ABB RAPID module: FSNH0464.mod

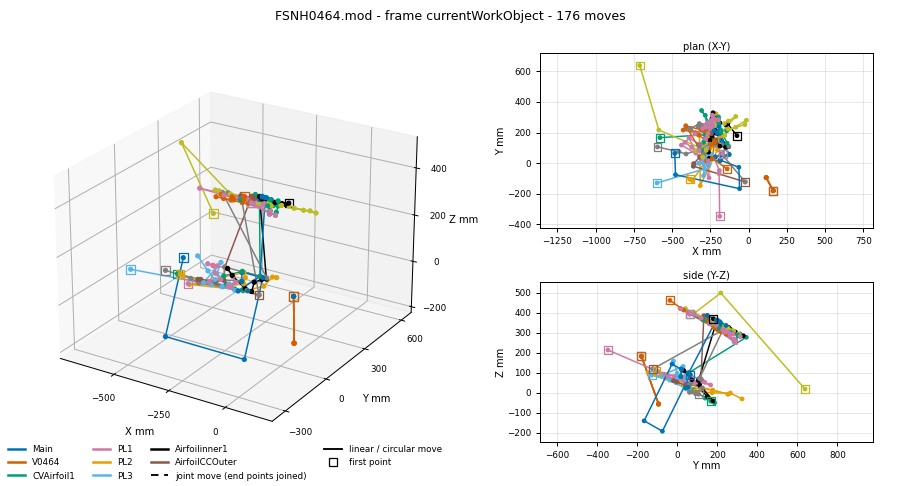
[picture p0: tool path of FSNH0464.mod in frame currentWorkObject, 176 of 176 moves have a stored position in this frame; points joined in program order, loops and branches not executed]
MODULE FSNH0464
    ! 10-10-24
    !
    ! declare and/or define variables that are local to this module
    LOCAL CONST listitem partProgram{3}:=[["","0464 Vane3"],["","Cooldown"],[stEmpty,"Stop"]];
    LOCAL VAR string defaultValueString;
    VAR num itemselected:=0;
    VAR buttondata buttonAnswer:=0;
    LOCAL VAR robtarget pInt_temp1;
	PERS zonedata pathairfoil:=[FALSE,100,100,100,75,75,15];
    !
    VAR num myTemp := 0;
    VAR num X_Shift := 0;
    VAR num X_Value := 0;
    VAR num Y_Shift := 0;
    VAR num Y_Value := 0;
    VAR num Z_Shift := 0;
    VAR num Z_Value := 0;
    VAR num Speed := 0;
    VAR num LargestDistance := 0;
    VAR num numberOfLines := 0;
    VAR num FirstPass := 0;
    !
    ! positions for Airfoil CTARR
    CONST robtarget p1:=[[-367.39,-113.29,109.00],[0.0618425,-0.927699,0.321538,0.179339],[-1,-1,-1,0],[0,120,9E+9,9E+9,9E+9,9E+9]];
    CONST robtarget p2:=[[-260.18,42.64,31.32],[0.0618425,-0.927699,0.321538,0.179339],[-1,-1,-1,0],[0,120,9E+9,9E+9,9E+9,9E+9]];
    CONST robtarget p3:=[[-238.83,117.01,17.08],[0.0618426,-0.927699,0.321538,0.179339],[-1,-1,-1,0],[0,120,9E+9,9E+9,9E+9,9E+9]];
    CONST robtarget p4:=[[-267.66,176.54,12.67],[0.0556447,-0.905315,0.344744,0.241786],[-1,-1,-1,0],[0,120,9E+9,9E+9,9E+9,9E+9]];
    CONST robtarget p5:=[[-321.65,253.11,-8.84],[0.063669,-0.890987,0.361532,0.267177],[-1,-1,-1,0],[0,120,9E+9,9E+9,9E+9,9E+9]];
    CONST robtarget p6:=[[1537.08,68.80,136.90],[0.258528,0.449073,0.847614,-0.114224],[0,0,0,0],[0,525.079,9E+9,9E+9,9E+9,9E+9]];
    CONST robtarget p7:=[[1532.27,28.26,128.24],[0.245924,0.528851,0.800385,-0.138642],[0,0,0,0],[0,558.621,9E+9,9E+9,9E+9,9E+9]];
    CONST robtarget p8:=[[-315.82,-146.53,99.01],[0.289971,-0.544816,0.776222,-0.128727],[0,0,0,0],[0,120,9E+9,9E+9,9E+9,9E+9]];
    CONST robtarget p9:=[[-204.02,86.23,8.60],[0.349716,-0.524325,0.773185,-0.0704735],[0,0,0,0],[0,120,9E+9,9E+9,9E+9,9E+9]];
    CONST robtarget p10:=[[-181.64,173.04,-1.69],[0.267612,-0.471353,0.840361,-0.00199147],[-1,0,0,0],[0,120,9E+9,9E+9,9E+9,9E+9]];
    !
    CONST robtarget p11:=[[-197.03,264.50,-2.50],[0.249749,-0.589134,0.759015,0.120175],[-1,-1,-1,0],[0,120,9E+9,9E+9,9E+9,9E+9]];
    CONST robtarget p12:=[[-213.54,323.24,-31.92],[0.254975,-0.617633,0.723692,0.172589],[-1,-1,-1,0],[0,120,9E+9,9E+9,9E+9,9E+9]];
    CONST robtarget p13:=[[1502.64,179.12,154.45],[0.27466,0.300473,0.910758,-0.0692597],[0,0,0,0],[0,525.079,9E+9,9E+9,9E+9,9E+9]];
    CONST robtarget p14:=[[1816.81,23.63,146.28],[0.530012,0.0601364,0.839977,0.0995457],[-1,0,-1,0],[0,485.704,9E+9,9E+9,9E+9,9E+9]];
    CONST robtarget p15:=[[1496.69,-77.72,540],[0.712477,-0.0505666,0.699591,0.0197792],[-1,-1,-1,0],[120.002,9E+09,9E+09,9E+09,9E+09,9E+09]];
    CONST robtarget p16:=[[1503.37,67.93,540],[0.712477,-0.0505667,0.699591,0.0197793],[-1,-1,-1,0],[150.003,9E+09,9E+09,9E+09,9E+09,9E+09]];
    CONST robtarget p17:=[[1525.14,108.88,540],[0.712477,-0.0505668,0.699591,0.0197793],[-1,-1,-1,0],[195.004,9E+09,9E+09,9E+09,9E+09,9E+09]];
    CONST robtarget p18:=[[1539.77,199.84,540],[0.712477,-0.0505668,0.699591,0.0197793],[-1,-1,-1,0],[230.001,9E+09,9E+09,9E+09,9E+09,9E+09]];
    CONST robtarget p19:=[[-192.48,-67.66,92.26],[0.242054,0.286611,0.916316,-0.140105],[0,1,0,0],[0,164,9E+9,9E+9,9E+9,9E+9]];
    CONST robtarget p20:=[[-191.44,-47.33,80.01],[0.242054,0.286612,0.916316,-0.140105],[0,1,0,0],[0,164,9E+9,9E+9,9E+9,9E+9]];
    !
    CONST robtarget p21:=[[-223.84,33.23,58.03],[0.242054,0.286612,0.916316,-0.140105],[0,1,0,0],[0,164,9E+9,9E+9,9E+9,9E+9]];
    CONST robtarget p22:=[[-271.49,90.03,49.56],[0.242053,0.286612,0.916315,-0.140105],[0,1,0,0],[0,164,9E+9,9E+9,9E+9,9E+9]];
    CONST robtarget p23:=[[-319.90,123.82,59.56],[0.242054,0.286612,0.916315,-0.140106],[0,1,0,0],[0,164,9E+9,9E+9,9E+9,9E+9]];
    CONST robtarget p24:=[[-390.01,166.06,37.60],[0.242053,0.286612,0.916315,-0.140106],[0,1,0,0],[0,164,9E+9,9E+9,9E+9,9E+9]];
    CONST robtarget p25:=[[1496.69,-77.72,650],[0.712477,-0.0505666,0.699591,0.0197792],[-1,-1,-1,0],[120.002,9E+09,9E+09,9E+09,9E+09,9E+09]];
    CONST robtarget p26:=[[-258.78,-95.71,104.93],[0.242054,0.286611,0.916316,-0.140105],[0,1,0,0],[0,164,9E+9,9E+9,9E+9,9E+9]];
    CONST robtarget p27:=[[-260.35,-14.42,80.84],[0.242054,0.286613,0.916315,-0.140105],[0,1,0,0],[0,164,9E+9,9E+9,9E+9,9E+9]];
    CONST robtarget p28:=[[-311.07,28.18,79.30],[0.242053,0.286612,0.916316,-0.140105],[0,1,0,0],[0,164,9E+9,9E+9,9E+9,9E+9]];
    CONST robtarget p29:=[[-344.71,65.79,87.67],[0.242054,0.286612,0.916315,-0.140106],[0,1,0,0],[0,164,9E+9,9E+9,9E+9,9E+9]];
    CONST robtarget p30:=[[-372.25,104.77,68.03],[0.242053,0.286612,0.916316,-0.140106],[0,1,0,0],[0,164,9E+9,9E+9,9E+9,9E+9]];
    !
    CONST robtarget p31:=[[-415.78,135.99,51.94],[0.242053,0.286612,0.916316,-0.140106],[0,1,0,0],[0,164,9E+9,9E+9,9E+9,9E+9]];
    CONST robtarget p32:=[[1621.31,158.58,690],[0.712477,-0.0505667,0.699591,0.0197792],[-1,-1,-1,0],[-0.00322896,9E+09,9E+09,9E+09,9E+09,9E+09]];
    CONST robtarget p33:=[[1620.84,58.68,700],[0.712477,-0.0505667,0.699591,0.0197793],[-1,-1,-1,0],[9.9958,9E+09,9E+09,9E+09,9E+09,9E+09]];
    CONST robtarget p34:=[[1665.7,-160.7,700],[0.712477,-0.0505667,0.699591,0.0197793],[-1,-1,-1,0],[70.0029,9E+09,9E+09,9E+09,9E+09,9E+09]];
    CONST robtarget p35:=[[1496.69,-77.72,700],[0.712477,-0.0505666,0.699591,0.0197792],[-1,-1,-1,0],[120.002,9E+09,9E+09,9E+09,9E+09,9E+09]];
    CONST robtarget p36:=[[1503.37,67.93,690],[0.712477,-0.0505667,0.699591,0.0197793],[-1,-1,-1,0],[150.003,9E+09,9E+09,9E+09,9E+09,9E+09]];
    CONST robtarget p37:=[[1525.14,108.88,690],[0.712477,-0.0505668,0.699591,0.0197793],[-1,-1,-1,0],[195.004,9E+09,9E+09,9E+09,9E+09,9E+09]];
    CONST robtarget p38:=[[1539.77,199.84,700],[0.712477,-0.0505668,0.699591,0.0197793],[-1,-1,-1,0],[230.001,9E+09,9E+09,9E+09,9E+09,9E+09]];
    CONST robtarget p39:=[[1444.86,284.59,700],[0.712477,-0.0505668,0.699591,0.0197793],[0,-1,-1,0],[270.004,9E+09,9E+09,9E+09,9E+09,9E+09]];
    CONST robtarget p40:=[[-288.13,-37.31,61.85],[0.0193858,-0.784247,0.616476,0.0673648],[-1,-1,-1,0],[0,102,9E+9,9E+9,9E+9,9E+9]];
    !
    CONST robtarget p41:=[[-241.42,56.91,12.34],[0.147864,-0.786015,0.586023,0.129978],[-1,-1,-1,0],[0,75,9E+9,9E+9,9E+9,9E+9]];
    CONST robtarget p42:=[[-266.80,56.10,32.67],[0.264437,-0.592967,0.760045,-0.0281851],[-1,-1,0,0],[0,6,9E+9,9E+9,9E+9,9E+9]];
    CONST robtarget p43:=[[-313.76,42.24,69.95],[0.310659,-0.477606,0.815293,-0.103346],[0,0,0,0],[0,-42,9E+9,9E+9,9E+9,9E+9]];
    CONST robtarget p44:=[[-285.87,28.41,130.28],[0.31066,-0.477606,0.815293,-0.103346],[0,0,0,0],[0,-78,9E+9,9E+9,9E+9,9E+9]];
    CONST robtarget p45:=[[-102.95,296.65,-15.64],[0.0526432,0.915175,-0.21481,-0.336957],[-1,-1,-1,0],[0,75,9E+9,9E+9,9E+9,9E+9]];
    CONST robtarget p46:=[[1762.50,190.04,67.00],[0.281257,0.841793,0.460433,0.0167615],[0,1,-1,0],[0,350,9E+9,9E+9,9E+9,9E+9]];
    CONST robtarget p48:=[[-294.40,-81.42,86.07],[0.12939,0.76137,-0.635239,0.00667964],[-1,-1,-1,0],[0,102,9E+9,9E+9,9E+9,9E+9]];
    CONST robtarget p49:=[[-258.19,-6.56,49.25],[0.0791781,0.771598,-0.630892,-0.0184961],[-1,-1,-1,0],[0,75,9E+9,9E+9,9E+9,9E+9]];

    PERS robtarget p201:=[[-158.45,259.15,313.28],[0.659486,-0.28722,0.405018,0.564396],[-1,1,-2,0],[0,-306.3,9E+9,9E+9,9E+9,9E+9]];
    PERS robtarget p202:=[[-208.97,252.93,315.49],[0.659485,-0.28722,0.405019,0.564397],[-1,1,-2,0],[0,-283.7,9E+9,9E+9,9E+9,9E+9]];
    PERS robtarget p203:=[[-236.09,220.83,319.38],[0.637208,-0.319422,0.454355,0.534319],[-1,1,-2,0],[0,-257.3,9E+9,9E+9,9E+9,9E+9]];
    PERS robtarget p204:=[[-344.66,82.28,398.40],[0.651502,-0.299469,0.423764,0.553432],[-1,1,-2,0],[0,-237.9,9E+9,9E+9,9E+9,9E+9]];
    PERS robtarget p205:=[[-138.38,318.26,282.97],[0.820959,-0.00154933,0.553533,0.14009],[0,2,-2,0],[0,-333.4,9E+9,9E+9,9E+9,9E+9]];
    PERS robtarget p206:=[[1522.85,30.49,127.90],[0.693528,-0.018539,0.719901,0.0204515],[-1,-1,-1,0],[0,525.079,9E+9,9E+9,9E+9,9E+9]];
    PERS robtarget p207:=[[1533.71,58.37,146.07],[0.688077,-0.0919601,0.714028,0.0908723],[-1,-1,-1,0],[0,525.079,9E+9,9E+9,9E+9,9E+9]];
    PERS robtarget p208:=[[-14.36,281.00,306.00],[0.489689,-0.400457,0.361391,0.685008],[-1,1,-2,0],[0,-338.2,9E+9,9E+9,9E+9,9E+9]];
    PERS robtarget p209:=[[-24.17,252.21,323.01],[0.489688,-0.400457,0.36139,0.685008],[-1,1,-2,0],[0,-321.5,9E+9,9E+9,9E+9,9E+9]];
    PERS robtarget p210:=[[-84.48,234.63,326.58],[0.659486,-0.28722,0.405018,0.564396],[-1,1,-2,0],[0,-306.3,9E+9,9E+9,9E+9,9E+9]];
    !
    PERS robtarget p211:=[[-133.52,222.77,331.59],[0.659485,-0.28722,0.405019,0.564397],[-1,1,-2,0],[0,-283.7,9E+9,9E+9,9E+9,9E+9]];
    PERS robtarget p212:=[[-155.56,181.99,339.83],[0.637208,-0.319422,0.454355,0.534319],[-1,1,-2,0],[0,-257.3,9E+9,9E+9,9E+9,9E+9]];
    PERS robtarget p213:=[[-300.90,40.20,419.83],[0.651502,-0.299469,0.423764,0.553432],[-1,1,-2,0],[0,-237.9,9E+9,9E+9,9E+9,9E+9]];
    PERS robtarget p214:=[[1526.81,49.01,147.72],[0.53358,0.309144,0.772491,-0.151589],[0,0,0,0],[0,525.079,9E+9,9E+9,9E+9,9E+9]];
    PERS robtarget p215:=[[-141.45,-101.58,920.03],[0.650986,0.194184,0.706774,-0.197436],[-1,0,0,0],[82.817,9E+09,9E+09,9E+09,9E+09,9E+09]];
    PERS robtarget p216:=[[-88.05,-18.09,920.70],[0.650993,0.194178,0.706763,-0.197458],[0,0,0,0],[82.817,9E+09,9E+09,9E+09,9E+09,9E+09]];
    PERS robtarget p217:=[[-21.87,98.95,918.25],[0.65099,0.194168,0.706777,-0.197427],[0,0,0,0],[82.817,9E+09,9E+09,9E+09,9E+09,9E+09]];
    PERS robtarget p218:=[[53.24,222.48,897.26],[0.65098,0.194179,0.706786,-0.197419],[0,0,0,0],[82.817,9E+09,9E+09,9E+09,9E+09,9E+09]];
    PERS robtarget p219:=[[45.58,94.46,899.85],[0.0855565,0.697288,0.707868,-0.0734352],[0,0,0,0],[104.005,9E+09,9E+09,9E+09,9E+09,9E+09]];
    PERS robtarget p220:=[[-237.32,31.15,412.31],[0.836251,-0.294327,0.277859,0.369933],[-1,2,-2,0],[0,-201.3,9E+9,9E+9,9E+9,9E+9]];
    !
    PERS robtarget p221:=[[-221.45,140.53,358.81],[0.836251,-0.294327,0.277859,0.369933],[-1,2,-2,0],[0,-201.3,9E+9,9E+9,9E+9,9E+9]];
    PERS robtarget p222:=[[-276.31,213.00,312.05],[0.822381,-0.324559,0.302501,0.356151],[-1,2,-3,0],[0,-201.3,9E+9,9E+9,9E+9,9E+9]];
    PERS robtarget p223:=[[-307.17,217.22,306.52],[0.822381,-0.324559,0.302501,0.356151],[0,2,-3,0],[0,-201.3,9E+9,9E+9,9E+9,9E+9]];
    PERS robtarget p224:=[[-410.54,245.03,291.11],[0.822381,-0.324559,0.302501,0.356151],[0,2,-3,0],[0,-201.3,9E+9,9E+9,9E+9,9E+9]];
    PERS robtarget p225:=[[1592.55,118.23,690.06],[0.505886,-0.101083,0.218555,-0.828308],[0,-1,1,0],[49.9958,9E+9,9E+9,9E+9,9E+9,9E+9]];
    PERS robtarget p226:=[[1608.55,16.90,696.10],[0.496587,-0.139785,0.281765,-0.808993],[0,-1,1,0],[25.0035,9E+9,9E+9,9E+9,9E+9,9E+9]];
    PERS robtarget p227:=[[1502.42,-81.35,694.68],[0.496587,-0.139785,0.281765,-0.808993],[0,-1,1,0],[0,9E+9,9E+9,9E+9,9E+9,9E+9]];
    PERS robtarget p228:=[[1461.90,-160.07,687.75],[0.496587,-0.139785,0.281765,-0.808993],[0,-1,1,0],[-0.000826709,9E+9,9E+9,9E+9,9E+9,9E+9]];
    !
    PERS robtarget p231:=[[-326.43,183.78,325.57],[0.822381,-0.324559,0.302501,0.356151],[0,2,-3,0],[0,-201.3,9E+9,9E+9,9E+9,9E+9]];
    PERS robtarget p232:=[[-347.83,199.42,314.58],[0.822381,-0.324559,0.302501,0.356151],[0,2,-3,0],[0,-201.3,9E+9,9E+9,9E+9,9E+9]];
    PERS robtarget p233:=[[-427.36,216.59,304.81],[0.822381,-0.324559,0.302501,0.35615],[0,2,-3,0],[0,-201.3,9E+9,9E+9,9E+9,9E+9]];
    PERS robtarget p234:=[[1381.21,176.71,690.45],[0.509919,-0.0782388,0.181097,-0.837296],[0,-1,1,0],[74.9967,9E+9,9E+9,9E+9,9E+9,9E+9]];
    PERS robtarget p235:=[[1460.37,118.23,690.06],[0.505886,-0.101083,0.218555,-0.828308],[0,-1,1,0],[49.9958,9E+9,9E+9,9E+9,9E+9,9E+9]];
    PERS robtarget p236:=[[1453.88,16.90,696.10],[0.496587,-0.139785,0.281765,-0.808993],[0,-1,1,0],[25.0035,9E+9,9E+9,9E+9,9E+9,9E+9]];
    PERS robtarget p237:=[[1308.94,-160.07,687.75],[0.496587,-0.139785,0.281765,-0.808993],[0,-1,1,0],[-0.000826709,9E+9,9E+9,9E+9,9E+9,9E+9]];
    PERS robtarget p238:=[[1411.45,-160.07,687.75],[0.496587,-0.139785,0.281765,-0.808993],[0,-1,1,0],[-0.000826709,9E+9,9E+9,9E+9,9E+9,9E+9]];
    !
    PERS robtarget p241:=[[1858.30,301.74,499.76],[0.179089,0.917392,0.34153,0.0983641],[0,1,0,0],[-175.061,9E+9,9E+9,9E+9,9E+9,9E+9]];
    PERS robtarget p242:=[[1614.86,199.00,509.29],[0.175594,0.951771,0.23609,0.086952],[0,1,-1,0],[-190.061,9E+9,9E+9,9E+9,9E+9,9E+9]];
    PERS robtarget p243:=[[1502.55,134.04,503.05],[0.185136,0.908581,0.362955,0.0920279],[0,1,0,0],[-220.061,9E+9,9E+9,9E+9,9E+9,9E+9]];
    PERS robtarget p244:=[[1494.58,104.81,490.86],[0.174159,0.800358,0.560783,0.120907],[0,1,0,0],[-240.061,9E+9,9E+9,9E+9,9E+9,9E+9]];
    PERS robtarget p245:=[[1559.49,159.93,488.36],[0.149738,0.674434,0.699604,0.182406],[0,1,0,0],[-310.061,9E+9,9E+9,9E+9,9E+9,9E+9]];
    PERS robtarget p246:=[[1600.54,33.00,493.44],[0.172748,0.593565,0.769913,0.158344],[-1,0,0,0],[-330.061,9E+9,9E+9,9E+9,9E+9,9E+9]];
    PERS robtarget p247:=[[1500.24,-78.88,512.52],[0.130233,0.625317,0.75886,0.12708],[-1,0,0,0],[-350.061,9E+9,9E+9,9E+9,9E+9,9E+9]];
    PERS robtarget p248:=[[1338.41,-93.31,512.24],[0.126705,0.803062,0.571687,0.110503],[-1,1,0,0],[-375.061,9E+9,9E+9,9E+9,9E+9,9E+9]];
    !

    ! declare and/or define position variables that are local to this module
	CONST robtarget home:=[[114.84,-94.02,-57.43],[0.398229,-0.576485,0.66735,0.252432],[-1,-1,-1,0],[0,372.2,9E+9,9E+9,9E+9,9E+9]];
	CONST robtarget pounce:=[[114.84,-94.02,-57.43],[0.398229,-0.576485,0.66735,0.252432],[-1,-1,-1,0],[0,0,9E+9,9E+9,9E+9,9E+9]];
    CONST robtarget home10:=[[-37.25,141.01,1171.15],[0.656992,0.226174,0.64921,-0.309408],[0,-1,0,0],[-0.00177226,9E+09,9E+09,9E+09,9E+09,9E+09]];
    PERS robtarget home20:=[[-47.87,162.56,920.76],[0.566373,0.264704,0.729584,-0.277237],[0,0,0,0],[0.0306373,9E+09,9E+09,9E+09,9E+09,9E+09]];
    PERS robtarget pounce10:=[[1506.92,-117.30,148.10],[0.362896,-0.228602,0.902396,0.0415831],[-1,-1,-1,0],[0,-6.2069,9E+9,9E+9,9E+9,9E+9]];
    PERS robtarget mypounce:=[[-385.16,-104.50,108.12],[0.0213445,-0.946834,0.217642,0.23597],[-1,-1,-1,0],[0,120,9E+9,9E+9,9E+9,9E+9]];
    PERS robtarget mypounce10:=[[-189.13,-347.09,212.55],[0.208106,0.294995,0.915526,-0.177429],[-1,1,0,0],[0,164,9E+9,9E+9,9E+9,9E+9]];
    PERS robtarget mypounce20:=[[-598.19,-128.68,86.61],[0.214705,-0.689144,0.690703,0.0437212],[0,-1,0,0],[0,75,9E+9,9E+9,9E+9,9E+9]];
    PERS robtarget mypounce30:=[[-579.47,167.00,-43.52],[0.403174,-0.614096,0.639379,0.227004],[0,-1,0,0],[0,-24.7,9E+9,9E+9,9E+9,9E+9]];
    PERS robtarget mypounce40:=[[-76.25,179.96,369.06],[0.403174,-0.614096,0.639379,0.227004],[-1,-1,-1,0],[0,-24.7,9E+9,9E+9,9E+9,9E+9]];
    PERS robtarget mypounce50:=[[-22.45,-122.19,118.26],[0.403174,-0.614096,0.639379,0.227004],[-1,-1,0,0],[0,-195,9E+9,9E+9,9E+9,9E+9]];
    PERS wobjdata wobj1:=[FALSE,TRUE,"",[[0,0,0],[1,0,0,0]],[[1526.4,-255.043,47.4813],[0.766931,0.185105,-0.133095,-0.599865]]];
    PERS robtarget p0:=[[1402.40,207.74,74.69],[0.420282,-0.489062,0.761608,-0.0643041],[0,-1,0,0],[0,453.104,9E+9,9E+9,9E+9,9E+9]];
    PERS robtarget mypounce60:=[[-595.25,106.44,-8.73],[0.422742,-0.506784,0.679012,0.321562],[0,1,-2,0],[0,-282,9E+9,9E+9,9E+9,9E+9]];
    PERS robtarget tempval:=[[1776.74,50.33,181.37],[0.419919,-0.484892,0.74874,-0.167142],[-1,-1,0,0],[0,453.104,9E+9,9E+9,9E+9,9E+9]];
    PERS robtarget tempval10:=[[1776.74,50.33,181.37],[0.419919,-0.484892,0.74874,-0.167142],[-1,-1,0,0],[0,453.104,9E+9,9E+9,9E+9,9E+9]];
    PERS robtarget mypouncePL:=[[1450.05,-296.49,158.45],[0.000887637,0.674822,0.737972,0.00347664],[-1,0,0,0],[0,368.4,9E+9,9E+9,9E+9,9E+9]];
    PERS robtarget mypouncePL10:=[[1453.74,-212.15,169.09],[0.000887898,0.674822,0.737972,0.00347632],[-1,0,0,0],[0,368.4,9E+9,9E+9,9E+9,9E+9]];
    PERS robtarget p50:=[[-294.93,-0.60,66.53],[0.062139,-0.617057,0.759744,-0.195367],[-1,-1,0,0],[0,6,9E+9,9E+9,9E+9,9E+9]];
    PERS robtarget p60:=[[-283.82,185.91,-51.33],[0.457128,-0.591319,0.607651,0.268583],[-1,-1,0,0],[0,-24.7,9E+9,9E+9,9E+9,9E+9]];
    PERS robtarget p70:=[[-239.02,202.70,360.69],[0.403174,-0.614096,0.639379,0.227004],[-1,-1,-1,0],[0,-24.7,9E+9,9E+9,9E+9,9E+9]];
    PERS robtarget p51:=[[-326.39,-0.73,96.25],[0.130195,-0.519879,0.792852,-0.290104],[0,0,0,0],[0,-42,9E+9,9E+9,9E+9,9E+9]];
    PERS robtarget p53:=[[8.76,359.17,-37.96],[0.0966582,0.980179,-0.140401,-0.100969],[-1,-1,-1,0],[0,75,9E+9,9E+9,9E+9,9E+9]];
    PERS robtarget p52:=[[-360.55,-19.52,158.17],[0.115329,-0.521701,0.78866,-0.304207],[0,0,0,0],[0,-78,9E+9,9E+9,9E+9,9E+9]];
    PERS robtarget p54:=[[1680.42,278.95,67.14],[0.281257,0.841793,0.460433,0.0167614],[0,1,-1,0],[0,350,9E+9,9E+9,9E+9,9E+9]];
    PERS robtarget p55:=[[1627.55,-144.85,103.80],[0.37608,-0.272238,0.874139,0.142592],[-1,-1,-1,0],[0,473.679,9E+9,9E+9,9E+9,9E+9]];
    PERS robtarget p56:=[[1636.24,-58.87,104.20],[0.37057,-0.304807,0.863301,0.156466],[-1,-1,-1,0],[0,473.679,9E+9,9E+9,9E+9,9E+9]];
    PERS robtarget p57:=[[1542.81,-38.49,90.01],[0.365729,-0.330862,0.853641,0.167539],[-1,-1,-1,0],[0,473.679,9E+9,9E+9,9E+9,9E+9]];
    PERS robtarget p58:=[[1415.80,3.28,64.46],[0.365729,-0.330862,0.853641,0.167539],[-1,-1,-1,0],[0,473.679,9E+9,9E+9,9E+9,9E+9]];
    PERS robtarget p67:=[[-307.25,344.42,276.28],[0.426614,-0.604806,0.62625,0.244992],[-1,-1,0,0],[0,-24.7,9E+9,9E+9,9E+9,9E+9]];
    PERS robtarget p61:=[[-292.56,138.30,-27.78],[0.451266,-0.594032,0.611365,0.264041],[-1,-1,0,0],[0,-24.7,9E+9,9E+9,9E+9,9E+9]];
    PERS robtarget p62:=[[-296.86,82.27,13.72],[0.403174,-0.614096,0.639379,0.227004],[-1,-1,0,0],[0,-24.7,9E+9,9E+9,9E+9,9E+9]];
    PERS robtarget p63:=[[-266.23,16.44,82.13],[0.403174,-0.614096,0.639379,0.227004],[-1,-1,0,0],[0,-24.7,9E+9,9E+9,9E+9,9E+9]];
    PERS robtarget p80:=[[-136.77,257.08,323.28],[0.403174,-0.614096,0.639379,0.227004],[-1,-1,-1,0],[0,-66.5,9E+9,9E+9,9E+9,9E+9]];
    PERS robtarget p81:=[[-148.29,250.44,326.38],[0.403174,-0.614096,0.639379,0.227004],[-1,-1,-1,0],[0,-66.5,9E+9,9E+9,9E+9,9E+9]];
    PERS robtarget p82:=[[-188.50,264.79,315.75],[0.474015,-0.57469,0.623128,0.238229],[-1,-1,0,0],[0,-66.5,9E+9,9E+9,9E+9,9E+9]];
    PERS robtarget p83:=[[-232.14,329.62,283.40],[0.321508,-0.678171,0.517716,0.410715],[-1,-1,-1,0],[0,-66.5,9E+9,9E+9,9E+9,9E+9]];
    PERS robtarget p93:=[[-257.39,31.23,110.38],[0.00262297,-0.734452,0.244527,0.633072],[-1,0,-2,0],[0,-66.5,9E+9,9E+9,9E+9,9E+9]];
    PERS robtarget p103:=[[-318.93,39.39,37.26],[0.627636,-0.216035,0.712765,-0.226646],[0,0,0,0],[0,-237,9E+9,9E+9,9E+9,9E+9]];
    PERS robtarget p94:=[[1375.79,-117.17,87.63],[0.605141,0.353098,0.62923,-0.336445],[0,0,-1,0],[0,525.079,9E+9,9E+9,9E+9,9E+9]];
    PERS robtarget p84:=[[-239.59,290.16,302.40],[0.155478,-0.729341,0.382687,0.545379],[-1,-1,-1,0],[0,-66.5,9E+9,9E+9,9E+9,9E+9]];
    PERS robtarget p85:=[[-215.79,212.41,343.83],[0.014859,-0.699079,0.252593,0.668778],[-1,0,-2,0],[0,-66.5,9E+9,9E+9,9E+9,9E+9]];
    PERS robtarget p95:=[[1571.42,84.90,94.72],[0.179969,0.647561,0.731941,-0.111974],[0,0,0,0],[0,368.4,9E+9,9E+9,9E+9,9E+9]];
    PERS robtarget p105:=[[-324.89,117.58,66.78],[0.416767,-0.646308,0.528374,0.359738],[-1,-1,0,0],[0,-195,9E+9,9E+9,9E+9,9E+9]];
    PERS robtarget p86:=[[-216.68,196.92,359.62],[0.00262296,-0.734452,0.244527,0.633072],[-1,0,-2,0],[0,-66.5,9E+9,9E+9,9E+9,9E+9]];
    PERS robtarget p87:=[[-130.30,108.22,66.21],[0.403174,-0.614096,0.639379,0.227004],[-1,-1,0,0],[0,-66.5,9E+9,9E+9,9E+9,9E+9]];
    PERS robtarget p97:=[[1571.42,84.90,94.72],[0.179969,0.647561,0.731941,-0.111974],[0,0,0,0],[0,368.4,9E+9,9E+9,9E+9,9E+9]];
    PERS robtarget p107:=[[-212.74,132.55,384.08],[0.65118,-0.247742,0.716886,0.0257505],[0,0,0,0],[0,-195,9E+9,9E+9,9E+9,9E+9]];
    PERS robtarget p88:=[[-150.48,105.12,60.16],[0.403174,-0.614096,0.639379,0.227004],[-1,-1,0,0],[0,-66.5,9E+9,9E+9,9E+9,9E+9]];
    PERS robtarget p89:=[[-187.38,111.78,37.90],[0.394279,-0.609579,0.66533,0.174051],[-1,-1,0,0],[0,-66.5,9E+9,9E+9,9E+9,9E+9]];
    PERS robtarget p68:=[[-283.10,312.74,292.50],[0.439315,-0.599378,0.618729,0.254799],[-1,-1,0,0],[0,-24.7,9E+9,9E+9,9E+9,9E+9]];
    PERS robtarget p59:=[[1256.15,38.08,77.18],[0.365729,-0.330862,0.853641,0.167539],[-1,-1,-1,0],[0,473.679,9E+9,9E+9,9E+9,9E+9]];
    PERS robtarget p47:=[[1532.27,28.26,128.24],[0.245924,0.528851,0.800385,-0.138642],[0,0,0,0],[0,558.621,9E+9,9E+9,9E+9,9E+9]];
    PERS robtarget p90:=[[-239.84,178.70,-41.54],[0.167334,-0.69714,0.619149,0.32039],[-1,-1,-1,0],[0,-66.5,9E+9,9E+9,9E+9,9E+9]];
    PERS robtarget p66:=[[1762.50,190.04,67.00],[0.281257,0.841793,0.460433,0.0167615],[0,1,-1,0],[0,350,9E+9,9E+9,9E+9,9E+9]];
    PERS robtarget p64:=[[-184.31,20.50,120.27],[0.421452,-0.606918,0.629232,0.241032],[-1,-1,0,0],[0,-24.7,9E+9,9E+9,9E+9,9E+9]];
    PERS robtarget p65:=[[-127.38,57.13,98.81],[0.403174,-0.614096,0.639379,0.227004],[-1,-1,0,0],[0,-24.7,9E+9,9E+9,9E+9,9E+9]];
    PERS robtarget p69:=[[-272.73,256.46,325.70],[0.403174,-0.614096,0.639379,0.227004],[-1,-1,-1,0],[0,-24.7,9E+9,9E+9,9E+9,9E+9]];
    PERS robtarget p71:=[[-182.89,218.68,346.20],[0.451214,-0.594056,0.611397,0.264],[-1,-1,-1,0],[0,-24.7,9E+9,9E+9,9E+9,9E+9]];
    PERS robtarget p72:=[[-142.49,211.94,352.22],[0.403174,-0.614096,0.639379,0.227004],[-1,-1,-1,0],[0,-24.7,9E+9,9E+9,9E+9,9E+9]];
    PERS robtarget p73:=[[1438.27,-226.26,170.27],[0.050777,0.553015,0.827359,-0.0840995],[-1,0,0,0],[0,350,9E+9,9E+9,9E+9,9E+9]];
    PERS robtarget home30:=[[160.81,-179.61,181.51],[0.375537,-0.58032,0.678284,0.24926],[-1,-1,-1,0],[0,0,9E+9,9E+9,9E+9,9E+9]];
    PERS robtarget mypounce70:=[[-586.63,217.02,497.85],[0.722927,-0.248634,0.347569,0.542912],[0,2,-2,0],[0,-295.1,9E+9,9E+9,9E+9,9E+9]];
    PERS robtarget p92:=[[-262.31,72.28,64.35],[0.0635228,0.75485,-0.188366,-0.625048],[-1,-1,-2,0],[0,-66.5,9E+9,9E+9,9E+9,9E+9]];
    PERS robtarget p102:=[[-358.96,-2.56,52.81],[0.63764,-0.102944,0.693172,-0.319892],[0,0,1,0],[0,-242,9E+9,9E+9,9E+9,9E+9]];
    PERS robtarget p91:=[[-251.62,150.06,-20.85],[0.139548,-0.838641,0.320424,0.417775],[-1,-1,-1,0],[0,-66.5,9E+9,9E+9,9E+9,9E+9]];
    PERS robtarget p100:=[[-162.78,-57.86,81.80],[0.585071,-0.326375,0.737712,-0.0833783],[0,0,0,0],[0,-188.2,9E+9,9E+9,9E+9,9E+9]];
    PERS robtarget p101:=[[-360.55,-19.69,59.35],[0.63764,-0.102945,0.693172,-0.319892],[0,0,1,0],[0,-245,9E+9,9E+9,9E+9,9E+9]];
    PERS robtarget p104:=[[-294.10,60.50,41.04],[0.612723,-0.440635,0.656029,-0.00611566],[0,-1,0,0],[0,-219,9E+9,9E+9,9E+9,9E+9]];
    PERS robtarget p106:=[[-129.79,110.40,70.28],[0.403174,-0.614096,0.639379,0.227004],[-1,-1,0,0],[0,-66.5,9E+9,9E+9,9E+9,9E+9]];
    PERS robtarget p108:=[[-211.79,151.68,368.97],[0.661248,-0.233352,0.711538,0.0448479],[0,0,0,0],[0,-195,9E+9,9E+9,9E+9,9E+9]];
    PERS robtarget p109:=[[-243.15,192.84,346.42],[0.574448,-0.491593,0.653442,0.0368712],[0,-1,0,0],[0,-195,9E+9,9E+9,9E+9,9E+9]];
    PERS robtarget p110:=[[-277.68,213.83,330.82],[0.505037,-0.583802,0.585982,0.24645],[-1,-1,0,0],[0,-195,9E+9,9E+9,9E+9,9E+9]];
    PERS robtarget p111:=[[-303.49,216.02,328.89],[0.416767,-0.646308,0.528374,0.359738],[-1,-1,-1,0],[0,-195,9E+9,9E+9,9E+9,9E+9]];
    PERS robtarget p112:=[[-329.18,242.61,321.09],[0.416767,-0.646308,0.528374,0.359738],[-1,-1,-1,0],[0,-195,9E+9,9E+9,9E+9,9E+9]];
    PERS robtarget p113:=[[-22.45,-122.19,118.26],[0.403174,-0.614096,0.639379,0.227004],[-1,-1,0,0],[0,-195,9E+9,9E+9,9E+9,9E+9]];
    PERS robtarget p123:=[[-250.95,124.67,23.71],[0.566357,-0.423499,0.622837,0.334608],[-1,1,-2,0],[0,-293,9E+9,9E+9,9E+9,9E+9]];
    PERS robtarget p120:=[[-454.95,74.33,3.15],[0.503111,-0.464695,0.606535,0.403798],[-1,1,-2,0],[0,-277.6,9E+9,9E+9,9E+9,9E+9]];
    PERS robtarget p121:=[[-408.85,60.36,0.80],[0.503111,-0.464695,0.606535,0.403798],[-1,1,-2,0],[0,-281.3,9E+9,9E+9,9E+9,9E+9]];
    PERS robtarget p131:=[[-407.31,65.48,14.57],[0.422742,-0.506784,0.679012,0.321562],[-1,1,-2,0],[0,-282,9E+9,9E+9,9E+9,9E+9]];
    PERS robtarget p122:=[[-319.61,90.88,-5.70],[0.606386,-0.392474,0.630174,0.284854],[0,1,-2,0],[0,-288,9E+9,9E+9,9E+9,9E+9]];
    PERS robtarget mypounce80:=[[-292.56,139.70,-25.36],[0.403174,-0.614096,0.639379,0.227004],[-1,-1,0,0],[0,-24,9E+9,9E+9,9E+9,9E+9]];
    PERS robtarget tp10:=[[-292.56,139.70,-25.36],[0.403174,-0.614096,0.639379,0.227004],[-1,-1,0,0],[0,-24,9E+9,9E+9,9E+9,9E+9]];
    !
    PERS robtarget mypounce110:=[[-482.41,64.04,89.43],[0.313843,-0.686244,0.567806,0.32889],[-1,-1,-1,0],[0,-31.4,9E+9,9E+9,9E+9,9E+9]];
    PERS robtarget p560:=[[-186.00,20.77,115.70],[0.313843,-0.686244,0.567806,0.32889],[-1,-1,-1,0],[0,-31.4,9E+9,9E+9,9E+9,9E+9]];
    PERS robtarget p561:=[[-186.00,20.77,115.70],[0.313843,-0.686244,0.567806,0.32889],[-1,-1,-1,0],[0,-24.7,9E+9,9E+9,9E+9,9E+9]];
    PERS robtarget p562:=[[-184.82,16.87,78.50],[0.313843,-0.686244,0.567806,0.32889],[-1,-1,-1,0],[0,6,9E+9,9E+9,9E+9,9E+9]];
    PERS robtarget p563:=[[-180.94,54.11,26.07],[0.313843,-0.686244,0.567806,0.32889],[-1,-1,-1,0],[0,60,9E+9,9E+9,9E+9,9E+9]];
    PERS robtarget p564:=[[-216.60,41.81,21.25],[0.313843,-0.686244,0.567806,0.32889],[-1,-1,-1,0],[0,108,9E+9,9E+9,9E+9,9E+9]];
    PERS robtarget p565:=[[-127.38,57.13,98.81],[0.403174,-0.614096,0.639379,0.227004],[-1,-1,0,0],[0,-24.7,9E+9,9E+9,9E+9,9E+9]];
    PERS robtarget p566:=[[-189.86,194.53,362.31],[0.403174,-0.614096,0.639379,0.227004],[-1,-1,-1,0],[0,-24.7,9E+9,9E+9,9E+9,9E+9]];
    PERS robtarget p569:=[[-194.35,212.02,353.83],[0.313843,-0.686244,0.567806,0.32889],[-1,-1,-1,0],[0,6,9E+9,9E+9,9E+9,9E+9]];
    PERS robtarget p567:=[[-175.65,149.52,386.03],[0.313843,-0.686244,0.567806,0.32889],[-1,-1,-1,0],[0,-31.4,9E+9,9E+9,9E+9,9E+9]];
    PERS robtarget p568:=[[-205.18,198.55,359.09],[0.313843,-0.686244,0.567806,0.32889],[-1,-1,-1,0],[0,-24.7,9E+9,9E+9,9E+9,9E+9]];
    PERS robtarget p570:=[[-192.85,243.24,335.35],[0.313843,-0.686244,0.567806,0.32889],[-1,-1,-1,0],[0,60,9E+9,9E+9,9E+9,9E+9]];
    PERS robtarget p571:=[[-228.38,214.17,338.21],[0.344401,-0.678774,0.547989,0.346931],[-1,-1,-1,0],[0,108,9E+9,9E+9,9E+9,9E+9]];
    PERS robtarget mypounce120:=[[-477.64,-74.92,-193.25],[0.313843,-0.686244,0.567806,0.32889],[-1,-1,0,0],[0,-31.4,9E+9,9E+9,9E+9,9E+9]];
    PERS robtarget mypounce130:=[[-59.04,-166.15,-141.34],[0.313843,-0.686244,0.567806,0.32889],[-1,-1,0,0],[0,-31.4,9E+9,9E+9,9E+9,9E+9]];
    PERS robtarget mypounce140:=[[-63.83,-26.70,142.30],[0.313843,-0.686244,0.567806,0.32889],[-1,-1,-1,0],[0,-31.4,9E+9,9E+9,9E+9,9E+9]];
    PERS robtarget mypounce90:=[[-284.25,-46.11,66.24],[0.0193857,-0.784247,0.616476,0.0673647],[-1,-1,-1,0],[0,102,9E+9,9E+9,9E+9,9E+9]];
    PERS robtarget p580:=[[-284.25,-46.11,66.24],[0.0193857,-0.784247,0.616476,0.0673647],[-1,-1,-1,0],[0,102,9E+9,9E+9,9E+9,9E+9]];
    PERS robtarget p589:=[[-284.25,-46.11,66.24],[0.0193857,-0.784247,0.616476,0.0673647],[-1,-1,-1,0],[0,102,9E+9,9E+9,9E+9,9E+9]];
    PERS robtarget p581:=[[-284.25,-46.11,66.24],[0.0193857,-0.784247,0.616476,0.0673647],[-1,-1,-1,0],[0,102,9E+9,9E+9,9E+9,9E+9]];
    PERS robtarget p582:=[[-284.25,-46.11,66.24],[0.0193857,-0.784247,0.616476,0.0673647],[-1,-1,-1,0],[0,102,9E+9,9E+9,9E+9,9E+9]];
    PERS robtarget p583:=[[-284.25,-46.11,66.24],[0.0193857,-0.784247,0.616476,0.0673647],[-1,-1,-1,0],[0,102,9E+9,9E+9,9E+9,9E+9]];
    PERS robtarget p584:=[[-284.25,-46.11,66.24],[0.0193857,-0.784247,0.616476,0.0673647],[-1,-1,-1,0],[0,102,9E+9,9E+9,9E+9,9E+9]];
    PERS robtarget p585:=[[-284.25,-46.11,66.24],[0.0193857,-0.784247,0.616476,0.0673647],[-1,-1,-1,0],[0,102,9E+9,9E+9,9E+9,9E+9]];
    PERS robtarget p586:=[[-284.25,-46.11,66.24],[0.0193857,-0.784247,0.616476,0.0673647],[-1,-1,-1,0],[0,102,9E+9,9E+9,9E+9,9E+9]];
    PERS robtarget p587:=[[-284.25,-46.11,66.24],[0.0193857,-0.784247,0.616476,0.0673647],[-1,-1,-1,0],[0,102,9E+9,9E+9,9E+9,9E+9]];
    PERS robtarget p588:=[[-284.25,-46.11,66.24],[0.0193857,-0.784247,0.616476,0.0673647],[-1,-1,-1,0],[0,102,9E+9,9E+9,9E+9,9E+9]];
    PERS robtarget p590:=[[-284.25,-46.11,66.24],[0.0193857,-0.784247,0.616476,0.0673647],[-1,-1,-1,0],[0,102,9E+9,9E+9,9E+9,9E+9]];
    PERS robtarget p591:=[[-284.25,-46.11,66.24],[0.0193857,-0.784247,0.616476,0.0673647],[-1,-1,-1,0],[0,102,9E+9,9E+9,9E+9,9E+9]];
    PERS robtarget p592:=[[-284.25,-46.11,66.24],[0.0193857,-0.784247,0.616476,0.0673647],[-1,-1,-1,0],[0,102,9E+9,9E+9,9E+9,9E+9]];
    PERS robtarget p593:=[[-284.25,-46.11,66.24],[0.0193857,-0.784247,0.616476,0.0673647],[-1,-1,-1,0],[0,102,9E+9,9E+9,9E+9,9E+9]];
    PERS robtarget mypounce100:=[[-277.25,84.01,395.93],[0.722927,-0.248634,0.347569,0.542912],[-1,1,-2,0],[0,-295.1,9E+9,9E+9,9E+9,9E+9]];
    PERS robtarget mypounce150:=[[-711.06,638.18,17.26],[0.631435,-0.398143,0.512601,0.424278],[0,2,-3,0],[0,-295.1,9E+9,9E+9,9E+9,9E+9]];
    PERS robtarget p126:=[[-408.23,232.10,321.99],[0.503111,-0.464695,0.606535,0.403798],[-1,1,-2,0],[0,-278.5,9E+9,9E+9,9E+9,9E+9]];
    PERS robtarget p127:=[[-377.53,226.81,328.68],[0.503111,-0.464695,0.606535,0.403798],[-1,1,-2,0],[0,-281.3,9E+9,9E+9,9E+9,9E+9]];
    PERS robtarget p128:=[[-321.81,258.79,307.10],[0.606386,-0.392473,0.630174,0.284853],[0,1,-2,0],[0,-288,9E+9,9E+9,9E+9,9E+9]];
    PERS robtarget p129:=[[-302.58,247.54,295.93],[0.589278,-0.408014,0.645554,0.263696],[0,1,-2,0],[0,-295.1,9E+9,9E+9,9E+9,9E+9]];
    PERS robtarget p251:=[[-131.76,239.79,323.25],[0.659486,-0.28722,0.405018,0.564396],[-1,1,-2,0],[0,-306.3,9E+9,9E+9,9E+9,9E+9]];
    PERS robtarget p261:=[[-131.76,239.79,323.25],[0.659486,-0.28722,0.405018,0.564396],[-1,1,-2,0],[0,-306.3,9E+9,9E+9,9E+9,9E+9]];
    PERS robtarget p200:=[[-132.29,275.77,309.60],[0.489688,-0.400457,0.36139,0.685008],[-1,1,-2,0],[0,-321.5,9E+9,9E+9,9E+9,9E+9]];
    PERS robtarget p199:=[[-84.16,305.60,292.73],[0.489689,-0.400457,0.361391,0.685008],[-1,1,-2,0],[0,-338.2,9E+9,9E+9,9E+9,9E+9]];
    PERS robtarget mypounce160:=[[-139.96,-36.96,460.48],[0.651502,-0.299469,0.423764,0.553432],[-1,1,-2,0],[0,-201.3,9E+9,9E+9,9E+9,9E+9]];
    PERS robtarget p229:=[[-274.30,15.45,419.41],[0.836251,-0.294327,0.277859,0.369933],[-1,2,-2,0],[0,-201.3,9E+9,9E+9,9E+9,9E+9]];
    PERS robtarget p230:=[[-241.32,121.35,367.90],[0.836251,-0.294327,0.277859,0.369933],[-1,2,-2,0],[0,-201.3,9E+9,9E+9,9E+9,9E+9]];
    PERS robtarget mypounce170:=[[-169.74,61.51,392.03],[0.631788,-0.302781,0.285021,0.654164],[-1,1,-2,0],[0,-108.095,9E+9,9E+9,9E+9,9E+9]];

    PERS robtarget p262:=[[-139.90,130.30,361.36],[0.589245,-0.359001,0.390168,0.609653],[-1,1,-2,0],[0,-108.095,9E+9,9E+9,9E+9,9E+9]];
    PERS robtarget p263:=[[-179.15,208.55,321.98],[0.589246,-0.359001,0.390168,0.609653],[-1,1,-2,0],[0,-101.595,9E+9,9E+9,9E+9,9E+9]];
    PERS robtarget p264:=[[-196.05,264.79,301.52],[0.601869,-0.414962,0.49282,0.4719],[-1,1,-2,0],[0,-83.0955,9E+9,9E+9,9E+9,9E+9]];
    PERS robtarget p265:=[[-196.91,303.11,286.35],[0.601868,-0.414962,0.49282,0.471901],[-1,1,-2,0],[0,-67.9955,9E+9,9E+9,9E+9,9E+9]];
    PERS robtarget p266:=[[-197.10,289.85,264.55],[0.547068,-0.46038,0.561521,0.416488],[-1,1,-2,0],[0,-67.9955,9E+9,9E+9,9E+9,9E+9]];
    PERS robtarget p267:=[[-197.16,283.70,254.22],[0.5098,-0.485421,0.600263,0.379677],[-1,0,-2,0],[0,-67.9955,9E+9,9E+9,9E+9,9E+9]];
    PERS robtarget p268:=[[-280.27,160.89,343.95],[0.589245,-0.359001,0.390168,0.609653],[-1,1,-2,0],[0,-108.095,9E+9,9E+9,9E+9,9E+9]];
    PERS robtarget p269:=[[-279.76,234.38,307.58],[0.570077,-0.361236,0.388648,0.627275],[-1,1,-2,0],[0,-101.595,9E+9,9E+9,9E+9,9E+9]];
    PERS robtarget p270:=[[-244.86,278.18,294.11],[0.400182,-0.465909,0.446248,0.650881],[-1,1,-2,0],[0,-83.0955,9E+9,9E+9,9E+9,9E+9]];
    PERS robtarget p271:=[[-235.76,313.49,280.59],[0.440871,-0.459023,0.457761,0.620794],[-1,1,-2,0],[0,-67.9955,9E+9,9E+9,9E+9,9E+9]];
    PERS robtarget p272:=[[-221.63,283.87,267.08],[0.43585,-0.50827,0.52651,0.523913],[-1,0,-2,0],[0,-67.9955,9E+9,9E+9,9E+9,9E+9]];
    PERS robtarget p273:=[[-228.94,291.69,249.76],[0.413617,-0.536087,0.563378,0.47343],[-1,0,-1,0],[0,-67.9955,9E+9,9E+9,9E+9,9E+9]];

    PERS robtarget p290:=[[-438.92,118.41,372.25],[0.526383,-0.32401,0.431914,0.656802],[-1,1,-2,0],[0,96.3057,9E+9,9E+9,9E+9,9E+9]];
    PERS robtarget p291:=[[-349.94,192.58,337.29],[0.526383,-0.324011,0.431914,0.656802],[-1,1,-2,0],[0,96.3057,9E+9,9E+9,9E+9,9E+9]];
    PERS robtarget p292:=[[-301.05,227.09,313.39],[0.496585,-0.350126,0.497544,0.619085],[-1,1,-2,0],[0,96.3057,9E+9,9E+9,9E+9,9E+9]];
    PERS robtarget p293:=[[-280.70,248.45,302.54],[0.420123,-0.397611,0.626384,0.522537],[-1,1,-2,0],[0,96.3057,9E+9,9E+9,9E+9,9E+9]];
    PERS robtarget p294:=[[-267.31,263.97,285.27],[0.385805,-0.412721,0.671645,0.479281],[-1,0,-2,0],[0,96.3057,9E+9,9E+9,9E+9,9E+9]];
    PERS robtarget p295:=[[-197.16,283.70,254.22],[0.5098,-0.485421,0.600263,0.379677],[-1,0,-2,0],[0,-67.9955,9E+9,9E+9,9E+9,9E+9]];
    PERS robtarget p296:=[[-280.27,160.89,343.95],[0.589245,-0.359001,0.390168,0.609653],[-1,1,-2,0],[0,-108.095,9E+9,9E+9,9E+9,9E+9]];
    PERS robtarget p297:=[[-279.76,234.38,307.58],[0.570077,-0.361236,0.388648,0.627275],[-1,1,-2,0],[0,-101.595,9E+9,9E+9,9E+9,9E+9]];
    PERS robtarget p298:=[[-244.86,278.18,294.11],[0.400182,-0.465909,0.446248,0.650881],[-1,1,-2,0],[0,-83.0955,9E+9,9E+9,9E+9,9E+9]];
    PERS robtarget p299:=[[-235.76,313.49,280.59],[0.440871,-0.459023,0.457761,0.620794],[-1,1,-2,0],[0,-67.9955,9E+9,9E+9,9E+9,9E+9]];
    PERS robtarget p300:=[[-324.02,83.31,391.45],[0.707426,-0.286817,0.430194,0.48189],[-1,1,-2,0],[0,96.3057,9E+9,9E+9,9E+9,9E+9]];
    PERS robtarget p301:=[[-265.68,194.75,337.64],[0.707426,-0.286817,0.430194,0.48189],[-1,1,-2,0],[0,96.3057,9E+9,9E+9,9E+9,9E+9]];
    PERS robtarget p302:=[[-251.98,230.69,312.45],[0.746771,-0.260149,0.494579,0.360621],[0,2,-2,0],[0,96.3057,9E+9,9E+9,9E+9,9E+9]];
    PERS robtarget p303:=[[-234.73,258.10,298.57],[0.621938,-0.281045,0.646804,0.340369],[0,1,-2,0],[0,96.3057,9E+9,9E+9,9E+9,9E+9]];
    PERS robtarget p304:=[[-243.68,236.60,302.54],[0.365798,-0.420186,0.695306,0.454077],[-1,0,-1,0],[0,96.3057,9E+9,9E+9,9E+9,9E+9]];
    PERS robtarget p305:=[[-228.94,291.69,249.76],[0.413617,-0.536087,0.563378,0.47343],[-1,0,-1,0],[0,-67.9955,9E+9,9E+9,9E+9,9E+9]];
    PERS robtarget p306:=[[-221.63,283.87,267.08],[0.43585,-0.50827,0.52651,0.523913],[-1,0,-2,0],[0,-67.9955,9E+9,9E+9,9E+9,9E+9]];
    PERS robtarget p307:=[[-228.94,291.69,249.76],[0.413617,-0.536087,0.563378,0.47343],[-1,0,-1,0],[0,-67.9955,9E+9,9E+9,9E+9,9E+9]];
    PERS robtarget p308:=[[-221.63,283.87,267.08],[0.43585,-0.50827,0.52651,0.523913],[-1,0,-2,0],[0,-67.9955,9E+9,9E+9,9E+9,9E+9]];
    PERS robtarget p309:=[[-228.94,291.69,249.76],[0.413617,-0.536087,0.563378,0.47343],[-1,0,-1,0],[0,-67.9955,9E+9,9E+9,9E+9,9E+9]];


    VAR num reg6:=0;
    VAR num reg7:=0;
    PERS robtarget mypounce180:=[[-264.32,16.76,418.93],[0.626936,-0.310345,0.298882,0.649082],[-1,1,-3,0],[0,96.3057,9E+9,9E+9,9E+9,9E+9]];

    !*************************************************************************************

    PROC Main()
	    !0464 Vane3\
        currentTool:=HVOF_375;
        currentWorkObject:=wobj1;
        !MoveAbsJ [[0,0,0,0,0,0],[0,0,0,0,0,0]]\NoEOffs, v1000, z50, currentTool\WObj:=currentWorkObject;

        TPErase;
        !prompt operator
        TPWrite "When Ready press 'Operator Start'";
        WaitDI DI_OP_Start, 1;
        TPErase;

        ! move to home position
        MoveL home30, v400, z10, currentTool\WObj:=currentWorkObject;

        ! get part program from operator
        itemSelected:=UIListView(\Result:=buttonAnswer,\Header:="FSNH_0464",partProgram,\Buttons:=btnOKCancel,\Icon:=iconInfo,\DefaultIndex:=1);

        IF buttonAnswer=resOK THEN
            IF itemSelected=1 THEN
              V0464;
            ELSEIF itemSelected=3 THEN
              Cooldown;
            ELSE
              GOTO StopCycle;
            ENDIF
        ELSE
            ! if user selects cancel then stop cycle
            GOTO StopCycle;
        ENDIF


        StopCycle:
        MoveL home30, v400, z10, currentTool\WObj:=currentWorkObject;

    ENDPROC


    PROC V0464()

	    ! set cycle counters
        coatingCycleCounter:=5;
        TPReadNum reg7, "how many heat passes?";

        ! allow operator to change the number of coating cycles from the default value
        defaultValueString := "default value = " + NumtoStr(coatingCycleCounter,0);
        coatingCycleCounter := UINumEntry (\Header:="Change Coating Cycles", \MsgArray:=["How many coating cycles?", defaultValueString], \InitValue:=coatingCycleCounter, \AsInteger);

        ! move to pounce position
        MoveJ home30, v800, z10, currentTool\WObj:=currentWorkObject;

        TPErase;
        TPWrite "Start Gun, and press 'Cycle Start' to Start";
        !
        WaitDI DI_OP_start, 1;
        TPErase;
        !heat passes
        IF reg7 > 0 THEN
            WHILE reg7>0 DO
              !
              PLATFORM;
              AIRFOIL;
              SHROUD;

              MoveL pounce, v800, z10, currentTool\WObj:=currentWorkObject;

              ! decrement the cycle counter
              reg7:=reg7-1;
              TPErase;
              TPWrite "number of coating cycles remaining = "\Num:=reg7;
              !
            ENDWHILE
        ENDIF

        MoveJ home30, v800, z10, currentTool\WObj:=currentWorkObject;
        !turn powder on
        TPWrite "Turn on powder, and press 'Cycle Start' to Start";
        !
        WaitDI DI_OP_start, 1;
        TPErase;
        MoveL pounce, v800, z10, currentTool\WObj:=currentWorkObject;

        WHILE coatingCycleCounter>0 DO
          !
          PLATFORM;
          AIRFOIL;
          SHROUD;

          MoveL pounce, v800, z10, currentTool\WObj:=currentWorkObject;

          ! decrement the cycle counter
          coatingCycleCounter:=coatingCycleCounter-1;
          TPErase;
          TPWrite "number of coating cycles remaining = "\Num:=coatingCycleCounter;
          !
        ENDWHILE
        !
        SKIP:
        !
        ! move to home position
        MoveL pounce, v800, z10, currentTool\WObj:=currentWorkObject;
        MoveL home30, v800, z10, currentTool\WObj:=currentWorkObject;

    ENDPROC

    !*************************************************************************************


    PROC AIRFOIL()
        !sprays Concave outer airfoil
        CVAirfoil1;
        Airfoilinner1;
        AirfoilCCOuter;
        Airlfoilinner2;
        !CTARCVAirfoil1;
    ENDPROC

    PROC SHROUD()
        !
        Shroud1;
        shroud2;
        Shroud3;
        Shroud4;
        !
    ENDPROC



    PROC PLATFORM()

        PL1;
        PL2;
        PL3;

        !
    ENDPROC


    PROC Cooldown()
		!
        !IF DI_Station_1 = 1 THEN
		!  rotateTable1AtSpeed 50;
        !ELSEIF DI_Station_2 = 1 THEN
		!  rotateTable2AtSpeed 50;
        !ENDIF
        !  WaitTime 300;
        !IF DI_Station_1 = 1 THEN
        !  stopTable1Rotation;
        !ELSEIF DI_Station_2 = 1 THEN
        !  stopTable2Rotation;
        !ENDIF
        !
        RETURN;
    ENDPROC

	PROC CVAirfoil1()
        MoveL mypounce30, v1000, z50, currentTool\WObj:=currentWorkObject;
        !MoveL tp10, v500, z1, currentTool\WObj:=currentWorkObject;
        SpeedFactors_3 5,5,5,5,5,5,5,5,5,5;
        SpeedFactors_4 5,5,5,5,5,5,5,5,5,5;

        Para4 5,500,60,67,6;

        RETURN;
        MoveL p60, v500, z1, currentTool\WObj:=currentWorkObject;
        MoveL p61, v500, z1, currentTool\WObj:=currentWorkObject;
		MoveL p62, v500, z1, currentTool\WObj:=currentWorkObject;
		MoveL p63, v500, z1, currentTool\WObj:=currentWorkObject;
		MoveL p64, v500, z1, currentTool\WObj:=currentWorkObject;
		MoveL p65, v500, z1, currentTool\WObj:=currentWorkObject;
		!MoveL p66, v500, z1, currentTool\WObj:=currentWorkObject;


		MoveL p67, v500, z1, currentTool\WObj:=currentWorkObject;
		MoveL p68, v500, z1, currentTool\WObj:=currentWorkObject;
		MoveL p69, v500, z1, currentTool\WObj:=currentWorkObject;
        MoveL p70, v500, z1, currentTool\WObj:=currentWorkObject;
        MoveL p71, v500, z1, currentTool\WObj:=currentWorkObject;
        MoveL p72, v500, z1, currentTool\WObj:=currentWorkObject;
        !MoveL p73, v500, z1, currentTool\WObj:=currentWorkObject;

		ENDPROC
	PROC PL1()
        MoveL mypounce10, v1000, z50, currentTool\WObj:=currentWorkObject;
        SpeedFactors_3 5,5,5,5,5,5,5,5,5,5;
        SpeedFactors_4 5,5,5,5,5,5,5,5,5,5;
        !Para3 5, 1000,50,52,53,55,3;
        Para4 5,500,19,26,6;
        !MoveL [[-486.61,-124.38,116.18],[0.0213445,-0.946834,0.217642,0.23597],[-1,-1,-1,0],[0,120,9E+9,9E+9,9E+9,9E+9]], v1000, z50, currentTool\WObj:=currentWorkObject;

        RETURN;
        MoveL p19, v1000, z50, currentTool\WObj:=currentWorkObject;
        MoveL p20, v1000, z50, currentTool\WObj:=currentWorkObject;
		MoveL p21, v500, z1, currentTool\WObj:=currentWorkObject;
		MoveL p22, v500, z1, currentTool\WObj:=currentWorkObject;
		MoveL p23, v500, z1, currentTool\WObj:=currentWorkObject;
		MoveL p24, v500, z1, currentTool\WObj:=currentWorkObject;
		!MoveL p25, v500, z1, currentTool\WObj:=currentWorkObject;

        MoveL p26, v500, z1, currentTool\WObj:=currentWorkObject;
		MoveL p27, v500, z1, currentTool\WObj:=currentWorkObject;
		MoveL p28, v500, z1, currentTool\WObj:=currentWorkObject;
		MoveL p29, v500, z1, currentTool\WObj:=currentWorkObject;
        MoveL p30, v500, z1, currentTool\WObj:=currentWorkObject;
        MoveL p31, v500, z1, currentTool\WObj:=currentWorkObject;
	ENDPROC
	PROC PL2()
        !inner platform
		MoveL mypounce, v1000, z50, currentTool\WObj:=currentWorkObject;
        SpeedFactors_3 5,5,5,5,5,5,5,5,5,5;
        SpeedFactors_4 5,5,5,5,5,5,5,5,5,5;
        !Para3 5, 1000,50,52,53,55,3;
        Para4 5,500,1,8,5;

        RETURN;
        MoveL p1, v1000, z50, currentTool\WObj:=currentWorkObject;
		MoveL p2, v500, z1, currentTool\WObj:=currentWorkObject;
		MoveL p3, v500, z1, currentTool\WObj:=currentWorkObject;
		MoveL p4, v500, z1, currentTool\WObj:=currentWorkObject;
		MoveL p5, v500, z1, currentTool\WObj:=currentWorkObject;
		!MoveL p6, v500, z1, currentTool\WObj:=currentWorkObject;
		!MoveL p7, v500, z1, currentTool\WObj:=currentWorkObject;

		MoveL p8, v500, z1, currentTool\WObj:=currentWorkObject;
		MoveL p9, v500, z1, currentTool\WObj:=currentWorkObject;
		MoveL p10, v500, z1, currentTool\WObj:=currentWorkObject;
        MoveL p11, v500, z1, currentTool\WObj:=currentWorkObject;
        MoveL p12, v500, z1, currentTool\WObj:=currentWorkObject;
	ENDPROC
	PROC PL3()
		MoveL mypounce20, v1000, z50, currentTool\WObj:=currentWorkObject;
        SpeedFactors_3 5,5,5,5,5,5,5,5,5,5;
        SpeedFactors_4 5,5,5,5,5,5,5,5,5,5;
        !Para3 5, 1000,50,52,53,55,3;
        Para4 5,500,40,48,5;
        RETURN;

        MoveL p40, v1000, z50, currentTool\WObj:=currentWorkObject;
        MoveL p41, v1000, z50, currentTool\WObj:=currentWorkObject;
		MoveL p42, v500, z1, currentTool\WObj:=currentWorkObject;
		MoveL p43, v500, z1, currentTool\WObj:=currentWorkObject;
		MoveL p44, v500, z1, currentTool\WObj:=currentWorkObject;
		!MoveL p45, v500, z1, currentTool\WObj:=currentWorkObject;
		!MoveL p46, v500, z1, currentTool\WObj:=currentWorkObject;


		MoveL p48, v500, z1, currentTool\WObj:=currentWorkObject;
		MoveL p49, v500, z1, currentTool\WObj:=currentWorkObject;
		MoveL p50, v500, z1, currentTool\WObj:=currentWorkObject;
        MoveL p51, v500, z1, currentTool\WObj:=currentWorkObject;
        MoveL p52, v500, z1, currentTool\WObj:=currentWorkObject;
        !MoveL p53, v500, z1, currentTool\WObj:=currentWorkObject;
        !MoveL p54, v500, z1, currentTool\WObj:=currentWorkObject;
	ENDPROC
	PROC Airfoilinner1()
        MoveL mypounce40, v1000, z50, currentTool\WObj:=currentWorkObject;
        SpeedFactors_3 5,5,5,5,5,5,5,5,5,5;
        SpeedFactors_4 5,5,5,5,5,5,5,5,5,5;

        Para4 5,500,80,87,7;

        RETURN;
        MoveL p80, v500, z1, currentTool\WObj:=currentWorkObject;
        MoveL p81, v500, z1, currentTool\WObj:=currentWorkObject;
		MoveL p82, v500, z1, currentTool\WObj:=currentWorkObject;
		MoveL p83, v500, z1, currentTool\WObj:=currentWorkObject;
		MoveL p84, v500, z1, currentTool\WObj:=currentWorkObject;
		MoveL p85, v500, z1, currentTool\WObj:=currentWorkObject;
		MoveL p86, v500, z1, currentTool\WObj:=currentWorkObject;

        MoveL p87, v500, z1, currentTool\WObj:=currentWorkObject;
		MoveL p88, v500, z1, currentTool\WObj:=currentWorkObject;
		MoveL p89, v500, z1, currentTool\WObj:=currentWorkObject;
		MoveL p90, v500, z1, currentTool\WObj:=currentWorkObject;
		MoveL p91, v500, z1, currentTool\WObj:=currentWorkObject;
        MoveL p92, v500, z1, currentTool\WObj:=currentWorkObject;
        MoveL p93, v500, z1, currentTool\WObj:=currentWorkObject;

		ENDPROC
	PROC AirfoilCCOuter()
        MoveL mypounce50, v1000, z50, currentTool\WObj:=currentWorkObject;
        SpeedFactors_3 6,6,6,6,6,6,6,6,6,6;
        SpeedFactors_4 6,6,6,6,6,6,6,6,6,6;

        Para4 5,500,101,107,5;

        RETURN;
        !MoveL p100, v500, z1, currentTool\WObj:=currentWorkObject;
        MoveL p101, v500, z1, currentTool\WObj:=currentWorkObject;
		MoveL p102, v500, z1, currentTool\WObj:=currentWorkObject;
		MoveL p103, v500, z1, currentTool\WObj:=currentWorkObject;
		MoveL p104, v500, z1, currentTool\WObj:=currentWorkObject;
		MoveL p105, v500, z1, currentTool\WObj:=currentWorkObject;
		!MoveL p106, v500, z1, currentTool\WObj:=currentWorkObject;

        MoveL p107, v500, z1, currentTool\WObj:=currentWorkObject;
		MoveL p108, v500, z1, currentTool\WObj:=currentWorkObject;
		MoveL p109, v500, z1, currentTool\WObj:=currentWorkObject;
		MoveL p110, v500, z1, currentTool\WObj:=currentWorkObject;
		MoveL p111, v500, z1, currentTool\WObj:=currentWorkObject;
        MoveL p112, v500, z1, currentTool\WObj:=currentWorkObject;
        !MoveL p113, v500, z1, currentTool\WObj:=currentWorkObject;
		ENDPROC
	PROC Airlfoilinner2()
		MoveL mypounce60, v1000, z50, currentTool\WObj:=currentWorkObject;
        SpeedFactors_3 6,6,6,6,6,6,6,6,6,6;
        SpeedFactors_4 6,6,6,6,6,6,6,6,6,6;

        Para4 5,500,120,126,4;

        RETURN;
        MoveL p120, v500, z1, currentTool\WObj:=currentWorkObject;
        MoveL p121, v500, z1, currentTool\WObj:=currentWorkObject;
		MoveL p122, v500, z1, currentTool\WObj:=currentWorkObject;
		MoveL p123, v500, z1, currentTool\WObj:=currentWorkObject;
		MoveL p104, v500, z1, currentTool\WObj:=currentWorkObject;
		MoveL p105, v500, z1, currentTool\WObj:=currentWorkObject;
		MoveL p106, v500, z1, currentTool\WObj:=currentWorkObject;

        MoveL p126, v500, z1, currentTool\WObj:=currentWorkObject;
		MoveL p127, v500, z1, currentTool\WObj:=currentWorkObject;
		MoveL p128, v500, z1, currentTool\WObj:=currentWorkObject;
		MoveL p129, v500, z1, currentTool\WObj:=currentWorkObject;
		MoveL p111, v500, z1, currentTool\WObj:=currentWorkObject;
        MoveL p112, v500, z1, currentTool\WObj:=currentWorkObject;
        MoveL p113, v500, z1, currentTool\WObj:=currentWorkObject;

	ENDPROC
	PROC Shroud1()
		MoveL mypounce150, v1000, z50, currentTool\WObj:=currentWorkObject;
		MoveL mypounce70, v1000, z50, currentTool\WObj:=currentWorkObject;
		MoveL mypounce100, v1000, z50, currentTool\WObj:=currentWorkObject;

        SpeedFactors_3 5,5,5,5,5,5,5,5,5,5;
        SpeedFactors_4 5,5,5,5,5,5,5,5,5,5;
        Para4 5,500,199,208,6;

        RETURN;
        MoveL p199, v500, z1, currentTool\WObj:=currentWorkObject;
        MoveL p200, v500, z1, currentTool\WObj:=currentWorkObject;
        MoveL p201, v500, z1, currentTool\WObj:=currentWorkObject;
        MoveL p202, v500, z1, currentTool\WObj:=currentWorkObject;
		MoveL p203, v500, z1, currentTool\WObj:=currentWorkObject;
		MoveL p204, v500, z1, currentTool\WObj:=currentWorkObject;
		!MoveL p205, v500, z1, currentTool\WObj:=currentWorkObject;
		!MoveL p206, v500, z1, currentTool\WObj:=currentWorkObject;
		!MoveL p207, v500, z1, currentTool\WObj:=currentWorkObject;

        MoveL p208, v500, z1, currentTool\WObj:=currentWorkObject;
		MoveL p209, v500, z1, currentTool\WObj:=currentWorkObject;
		MoveL p210, v500, z1, currentTool\WObj:=currentWorkObject;
		MoveL p211, v500, z1, currentTool\WObj:=currentWorkObject;
		MoveL p212, v500, z1, currentTool\WObj:=currentWorkObject;
        MoveL p213, v500, z1, currentTool\WObj:=currentWorkObject;
        !MoveL p214, v500, z1, currentTool\WObj:=currentWorkObject;


	ENDPROC
	PROC CTARCVAirfoil1()
		MoveL mypounce110, v1000, z50, currentTool\WObj:=currentWorkObject;
		MoveL mypounce120, v1000, z50, currentTool\WObj:=currentWorkObject;
		MoveL mypounce130, v1000, z50, currentTool\WObj:=currentWorkObject;
		MoveL mypounce140, v1000, z50, currentTool\WObj:=currentWorkObject;

        SpeedFactors_3 5,5,5,5,5,5,5,5,5,5;
        SpeedFactors_4 5,5,5,5,5,5,5,5,5,5;

        Para4 5,500,560,567,5;

        RETURN;
        MoveL p560, v500, z1, currentTool\WObj:=currentWorkObject;
        MoveL p561, v500, z1, currentTool\WObj:=currentWorkObject;
		MoveL p562, v500, z1, currentTool\WObj:=currentWorkObject;
		MoveL p563, v500, z1, currentTool\WObj:=currentWorkObject;
		MoveL p564, v500, z1, currentTool\WObj:=currentWorkObject;
		MoveL p565, v500, z1, currentTool\WObj:=currentWorkObject;
		MoveL p566, v500, z1, currentTool\WObj:=currentWorkObject;


		MoveL p567, v500, z1, currentTool\WObj:=currentWorkObject;
		MoveL p568, v500, z1, currentTool\WObj:=currentWorkObject;
		MoveL p569, v500, z1, currentTool\WObj:=currentWorkObject;
        MoveL p570, v500, z1, currentTool\WObj:=currentWorkObject;
        MoveL p571, v500, z1, currentTool\WObj:=currentWorkObject;

	ENDPROC

	PROC shroud2()
		MoveL mypounce160, v1000, z50, currentTool\WObj:=currentWorkObject;

        SpeedFactors_3 5,5,5,5,5,5,5,5,5,5;
        SpeedFactors_4 5,5,5,5,5,5,5,5,5,5;
        Para4 5,500,220,229,5;

        RETURN;
        MoveL p220, v500, z1, currentTool\WObj:=currentWorkObject;
        MoveL p221, v500, z1, currentTool\WObj:=currentWorkObject;
        MoveL p222, v500, z1, currentTool\WObj:=currentWorkObject;
        MoveL p223, v500, z1, currentTool\WObj:=currentWorkObject;
		MoveL p224, v500, z1, currentTool\WObj:=currentWorkObject;
		!MoveL p225, v500, z1, currentTool\WObj:=currentWorkObject;
		!MoveL p226, v500, z1, currentTool\WObj:=currentWorkObject;
		!MoveL p227, v500, z1, currentTool\WObj:=currentWorkObject;
		!MoveL p228, v500, z1, currentTool\WObj:=currentWorkObject;

        MoveL p229, v500, z1, currentTool\WObj:=currentWorkObject;
		MoveL p230, v500, z1, currentTool\WObj:=currentWorkObject;
		MoveL p231, v500, z1, currentTool\WObj:=currentWorkObject;
		MoveL p232, v500, z1, currentTool\WObj:=currentWorkObject;
		MoveL p233, v500, z1, currentTool\WObj:=currentWorkObject;
        !MoveL p234, v500, z1, currentTool\WObj:=currentWorkObject;
        !MoveL p235, v500, z1, currentTool\WObj:=currentWorkObject;

	ENDPROC
	PROC Shroud3()
		MoveL mypounce170, v1000, z50, currentTool\WObj:=currentWorkObject;

        SpeedFactors_3 5,5,5,5,5,5,5,5,5,5;
        SpeedFactors_4 5,5,5,5,5,5,5,5,5,5;
        Para4 5,500,262,268,6;

        RETURN;
        MoveL p262, v500, z1, currentTool\WObj:=currentWorkObject;
        MoveL p263, v500, z1, currentTool\WObj:=currentWorkObject;
        MoveL p264, v500, z1, currentTool\WObj:=currentWorkObject;
        MoveL p265, v500, z1, currentTool\WObj:=currentWorkObject;
		MoveL p266, v500, z1, currentTool\WObj:=currentWorkObject;
		MoveL p267, v500, z1, currentTool\WObj:=currentWorkObject;

        MoveL p268, v500, z1, currentTool\WObj:=currentWorkObject;
		MoveL p269, v500, z1, currentTool\WObj:=currentWorkObject;
		MoveL p270, v500, z1, currentTool\WObj:=currentWorkObject;
        MoveL p271, v500, z1, currentTool\WObj:=currentWorkObject;
		MoveL p272, v500, z1, currentTool\WObj:=currentWorkObject;
		MoveL p273, v500, z1, currentTool\WObj:=currentWorkObject;


	ENDPROC

    PROC Shroud4()
		MoveL mypounce170, v1000, z50, currentTool\WObj:=currentWorkObject;
		MoveL mypounce180, v1000, z50, currentTool\WObj:=currentWorkObject;

        SpeedFactors_3 5,5,7,7,7,5,5,5,5,5;
        SpeedFactors_4 5,5,5,5,5,5,5,5,5,5;
        Para4 5,500,290,300,5;

        RETURN;
        MoveL p290, v500, z1, currentTool\WObj:=currentWorkObject;
        MoveL p291, v500, z1, currentTool\WObj:=currentWorkObject;
        MoveL p292, v500, z1, currentTool\WObj:=currentWorkObject;
        MoveL p293, v500, z1, currentTool\WObj:=currentWorkObject;
		MoveL p294, v500, z1, currentTool\WObj:=currentWorkObject;
		MoveL p295, v500, z1, currentTool\WObj:=currentWorkObject;
        MoveL p296, v500, z1, currentTool\WObj:=currentWorkObject;
		MoveL p297, v500, z1, currentTool\WObj:=currentWorkObject;
		MoveL p298, v500, z1, currentTool\WObj:=currentWorkObject;
		MoveL p299, v500, z1, currentTool\WObj:=currentWorkObject;

        MoveL p300, v500, z1, currentTool\WObj:=currentWorkObject;
		MoveL p301, v500, z1, currentTool\WObj:=currentWorkObject;
        MoveL p302, v500, z1, currentTool\WObj:=currentWorkObject;
		MoveL p303, v500, z1, currentTool\WObj:=currentWorkObject;
		MoveL p304, v500, z1, currentTool\WObj:=currentWorkObject;
        MoveL p305, v500, z1, currentTool\WObj:=currentWorkObject;
		MoveL p306, v500, z1, currentTool\WObj:=currentWorkObject;
		MoveL p307, v500, z1, currentTool\WObj:=currentWorkObject;
		MoveL p308, v500, z1, currentTool\WObj:=currentWorkObject;
		MoveL p309, v500, z1, currentTool\WObj:=currentWorkObject;

	ENDPROC

ENDMODULE
